KUKA KRL program: vw_bn_usr_s.src, vw_bn_usr_s.dat

--- vw_bn_usr_s.src ---
&ACCESS RV
&REL 11
&COMMENT KS_1.0
&PARAM DISKPATH = KRC:\R1\VW_User\Applikation\Blindnietmuttern
&PARAM TPVW_VERSION = 8.1.8
DEF vw_bn_usr_s( )
;FOLD Aenderungsjournal
;*-------------------------------------------------*
;*Technologiepaket Blindnietmuttern                *
;*                                                 *
;*Konzernstandard                                  *
;*Bearbeiter: B.Mildenberger PEF-2/E0A             *
;*                                                 *
;* Erstellt am:                                    *
;* 2016.02.19 BM                                   *
;*                                                 *
;* Aenderungsjournal                               *
;*                                                 *
;*-------------------------------------------------*
;ENDFOLD Aenderungsjournal
END
;
;FOLD INIT Blindnietmuttern
GLOBAL DEF BN_INIT( )
INT i
;
;FOLD Version Techpaket
Tech_BN.Name[]="KS24.01.002_160220"
;ENDFOLD
;
;FOLD Vorbesetzung Meldungsausgabe
FOR I = 1 TO 100
  n_BN_Handle[I]=-1
ENDFOR
;ENDFOLD
;
$OUT[O_BN_StartPrz[1]]=FALSE
;
END
;ENDFOLD
;
;---------------------------------------------------
;FOLD SAW Blindnietmuttern
GLOBAL DEF BN_SAW( )
INT i
;
;
END
;ENDFOLD
;
;---------------------------------------------------
;FOLD RESET Blindnietmuttern
GLOBAL DEF BN_RESET( )
INT i
;
$OUT[O_BN_StartPrz[1]]=FALSE
;
END
;ENDFOLD
;
;---------------------------------------------------
;FOLD CANCEL Blindnietmuttern
GLOBAL DEF BN_CANCEL( )
INT i
;
$OUT[O_BN_StartPrz[1]]=FALSE
;
END
;ENDFOLD
;
;---------------------------------------------------
;FOLD LOOP Blindnietmuttern
GLOBAL DEF BN_LOOP()
;
FOR BN_ActApp = 1 TO BN_MaxApp
  IF Mit_BN[BN_ActApp] THEN
    ;FOLD Lebensbit
    BN_lBit(BN_ActApp)
    ;ENDFOLD Lebensbit
;
    ;RESET im Fehlerfall ausloesen
    IF NOT BN_QuitHifu[BN_ActApp] AND (NOT $OUT[O_R_SAK] OR NOT $OUT[O_R_RK100]) THEN
      BN_QuitHifu[BN_ActApp]=TRUE
      ;Anstehende Prozesse sicher beenden
      $OUT[O_BN_Reload[BN_ActApp]]=FALSE
      $OUT[O_BN_StartPrz[BN_ActApp]]=FALSE
    ENDIF
    SWITCH BN1_ErrorCode ;Gezieltes Quittieren selektierter Fehler
	  CASE 107, 108
	    BN_FrgQuitHifu[BN_ActApp]=FALSE;keine Freigabe Autoquit
	  DEFAULT
        BN_FrgQuitHifu[BN_ActApp]=TRUE
	ENDSWITCH
    ;Ruecksetzen Ausgaben nach Fehler
    IF $OUT[O_R_RK100] AND $OUT[O_R_SAK] AND BN_QuitHifu[BN_ActApp] AND BN_FrgQuitHifu[BN_ActApp] AND $COULD_START_MOTION THEN
      $OUT[O_BN_Reset[BN_ActApp]]=TRUE
	  IF (($ROB_TIMER - QuitTimer_BN[BN_ActApp]) > 500) THEN
	    $OUT[O_BN_Init[BN_ActApp]]=TRUE
	    $OUT[O_BN_Reset[BN_ActApp]]=FALSE
		IF $OUT[O_BN_Init[BN_ActApp]] AND $IN[I_BN_FkInit[BN_ActApp]] THEN
  	      $OUT[O_BN_Init[BN_ActApp]]=FALSE
		  BN_QuitHifu[BN_ActApp]=FALSE
	    ELSE
        IF (($ROB_TIMER - QuitTimer_BN[BN_ActApp]) > 5000) AND $IN[I_BN_AUTO[BN_ActApp]] THEN
		    BN_Msg(2,#QuitMsg)
			;Retry Init
			$OUT[O_BN_Reset[BN_ActApp]]=TRUE
			QuitTimer_BN[BN_ActApp] = 0
            QuitTimer_BN[BN_ActApp] = $ROB_TIMER
		  ENDIF
		ENDIF
	  ENDIF
	ELSE
      QuitTimer_BN[BN_ActApp] = 0
      QuitTimer_BN[BN_ActApp] = $ROB_TIMER
    ENDIF
;
    ;BA-Hand an BNx setzen
    IF $OUT[O_R_Hand] AND NOT $COULD_START_MOTION THEN
      $OUT[O_BN_R_Hand[BN_ActApp]]=TRUE
      $OUT[O_BN_R_Auto[BN_ActApp]]=FALSE
    ENDIF
;
    ;BA-AUTO an NZ 1 setzen
    IF ($OUT[O_R_Proz_akt] OR $OUT[O_R_bewegt]) OR $OUT[O_R_Auto] THEN
      $OUT[O_BN_R_Hand[BN_ActApp]]=FALSE
      $OUT[O_BN_R_Auto[BN_ActApp]]=TRUE
    ENDIF
;
    ;Anwahl Energiesparmodus
    $OUT[O_BN_eMode[BN_ActApp]] = (($Brake_Sig==0) AND $timer_flag[TimerNr_E_Mo] AND e_Mode_Hilf2)
    ;Freigabe Steuerluft
    $OUT[O_BN_FrgP[BN_ActApp]] = $IN[I_BD01ND] AND $IN[I_MedVorh]
;
    ;Setzweg fuer Visualisierung in CorrMode
	BN_Setzweg_Act[BN_ActApp]=ABS(BN1_SetzWeg)/10 ;[1/10mm]
;
    ;Ausgabe Fehlermeldungen
;
    ;Nieten n.i.O.
    $OUT[O_BN_PrzNio[BN_ActApp]]=$OUT[O_R_Auto] AND $COULD_START_MOTION AND $OUT[O_BN_P_act[BN_ActApp]] AND $FLAG[F_BN_PrzNiO[BN_ActApp]]
    ;Vorwarnung liegt an
    $OUT[O_BN_VwStdm[BN_ActApp]]=$OUT[O_R_Auto] AND $COULD_START_MOTION AND ($IN[I_BN_WarnZugDorn[BN_ActApp]] OR $IN[I_BN_WarnOel[BN_ActApp]])
    ;Verklemmanzeige
    $OUT[O_BN_Verkl[BN_ActApp]]=$OUT[O_R_Auto] AND $COULD_START_MOTION AND NOT $IN[I_BN_AusglIo[BN_ActApp]]
    ;Startbereit fehlt
    $OUT[O_BN_StartBerFehl[BN_ActApp]]=$OUT[O_R_Auto] AND $COULD_START_MOTION AND NOT $IN[I_BN_Ready[BN_ActApp]] AND $FLAG[F_BN_Sammel[BN_ActApp]] AND $timer_flag[TimerNr_Ein]
    ;Betriebsbereit fehlt
    $OUT[O_BN_BereitFehlt[BN_ActApp]]=$OUT[O_R_Auto] AND $COULD_START_MOTION AND NOT $IN[I_BN_Ready[BN_ActApp]] AND $timer_flag[TimerNr_Ein]
    ;Sammelstoerung
    $OUT[O_BN_Sammel[BN_ActApp]]=$OUT[O_R_Auto] AND $COULD_START_MOTION AND ($FLAG[F_BN_Sammel[BN_ActApp]] OR $IN[I_BN_Sammel[BN_ActApp]] OR BN_LBitFeh[BN_ActApp] OR $IN[I_BN_StdmZugDorn[BN_ActApp]]) AND $timer_flag[TimerNr_Ein]
    ;Stoerung quittieren
	IF (BN_ActApp==1) THEN
 	  BN_ErrorCodeAct[1]=BN1_ErrorCode
	ENDIF
	SWITCH BN1_ErrorCode ;Vorhaltung zur gezielten Reaktion auf bestimmte Fehleransprachen
	  CASE 0
	    ;löppt
	  CASE 108 ; Fehler Zugdorn darf nicht via Panel quittiert werden
	    ;#dummy
	  DEFAULT
        $OUT[O_BN_Reset[BN_ActApp]]= $IN[I_BN_Sammel[BN_ActApp]] AND $IN[I_BN_AnwZ1[BN_ActApp]] AND $IN[I_R_Quit_Wei]
	ENDSWITCH
;
    ;Ausgabe Zangencode
    IF NOT Docking THEN
      BN1_ZCode=1
    ENDIF
;
  ENDIF
ENDFOR
;
;ENDFOLD
END
;ENDFOLD
;
;---------------------------------------------------
;---------------------------------------------------
;FOLD Blindnietmuttern_Meldungen
DEF BN_Msg(msg_nr :IN, MsgTyp :IN)
INT msg_nr, Answer
DECL BN_MsgType MsgTyp
DECL KrlMsg_T USER_MSG
DECL KrlMsgPar_T Par[3]
DECL KrlMsgOpt_T Opt
;
USER_MSG = { Modul[] "BN_S_Msg", Nr -1, Msg_txt[] " "}
Opt = { VL_Stop FALSE, Clear_P_Reset TRUE, Log_To_DB TRUE }
Par[1] = { Par_type #Value, Par_txt[] " " }
;
;
IF ((n_BN_Handle[msg_nr]<0) OR (MsgTyp==#NotifyMsg) OR (MsgTyp==#QuitMsg)) THEN
  USER_MSG.Nr = msg_nr
  SWITCH msg_nr
    CASE 1
	   USER_MSG.MSG_TXT[]="Blindnietmutternsteuerung Lebensbitfehler"
    CASE 2
	   USER_MSG.MSG_TXT[]="Initialisierungsfehler Blindnietmutternsteuerung"
    DEFAULT
	   USER_MSG.MSG_TXT[]="unbekannte Meldung"
  ENDSWITCH
  SWITCH MsgTyp
    CASE #StateMsg
      n_BN_Handle[msg_nr] = Set_KrlMsg (#State, USER_MSG, Par[], Opt) ;Ausgabe Statusmeldung
    CASE #QuitMsg
      n_BN_Handle[msg_nr] = Set_KrlMsg (#Quit, USER_MSG, Par[], Opt) ;Ausgabe Quittierungsmeldung
    CASE #NotifyMsg
      n_BN_Handle[msg_nr] = Set_KrlMsg (#Notify, USER_MSG, Par[], Opt) ;Ausgabe Hinweismeldung
    DEFAULT
      n_BN_Handle[msg_nr] = Set_KrlMsg (#Quit, USER_MSG, Par[], Opt) ;Ausgabe Quittierungsmeldung
  ENDSWITCH
ENDIF
END
;
;ENDFOLD (Blindnietmuttern Meldungen)
;
;---------------------------------------------------
;FOLD Lebensbit Blindnietmuttern
DEF BN_lBit(AppNr:IN)
BOOL LBitBZ1, bRet
INT AppNr

BN_LBitFeh[AppNr]=FALSE
;Setzen - Rucksetzen Lebensbit Roboter
$OUT[O_BN_LBitRobBn[AppNr]]=NOT $IN[I_BN_LBitBnRob[AppNr]]
;Pruefen Lebensbit von BZ1
IF $IN[I_BN_LBitBnRob[AppNr]]==FALSE THEN
  IF LBitBnRem[AppNr]==FALSE THEN
    TimerNr_BN[AppNr]=$ROB_TIMER
  ENDIF
  LBitBnRem[AppNr]=TRUE
ELSE
  IF LBitBnRem[AppNr]==TRUE THEN
    TimerNr_BN[AppNr]=$ROB_TIMER
  ENDIF
  LBitBnRem[AppNr]=FALSE
ENDIF
;
IF ($ROB_TIMER - TimerNr_BN[AppNr]) > 5000 THEN
  BN_LBitFeh[AppNr]=TRUE
ENDIF
;
IF BN_LBitFeh[AppNr] THEN
  BN_Msg(1,#StateMsg)
ELSE
  BN_LBitFeh[AppNr]=FALSE
ENDIF
END
;ENDFOLD Lebensbit Blindnietmuttern
;

--- vw_bn_usr_s.dat ---
&ACCESS  RV
&COMMENT KS_1.0
&PARAM DISKPATH = VW_User/Applikation/Blindnietmuttern
&PARAM TPVW_VERSION = 8.1.8
&REL 11
DEFDAT  vw_bn_usr_s PUBLIC
;
;*-------------------------------------------------*
;*Technologiepaket Blindnietmuttern                *
;*                                                 *
;*Konzernstandard                                  *
;*Bearbeiter: B.Mildenberger PEF-2/E0A             *
;*                                                 *
;* Erstellt am:                                    *
;* 2016.02.19 BM                                   *
;*                                                 *
;* Aenderungsjournal                               *
;*                                                 *
;*-------------------------------------------------*
;
;FOLD USER_Version
STRUC _Tech_BN CHAR Name[20],INT Datum
DECL _Tech_BN Tech_BN
;ENDFOLD USER_VERSION
;
;FOLD Vorwahlen
GLOBAL BOOL MIT_BN[1]
MIT_BN[1]=FALSE
;ENDFOLD Vorwahlen
;
;FOLD Stukturen
;
;ENDFOLD Strukturen
;
;FOLD Flags
GLOBAL INT F_m_BN[1]
F_m_BN[1]=422
;ENDFOLD FLAGS
;
;FOLD BOOLEAN
;
GLOBAL BOOL LBitBnRem[1]
LBitBnRem[1]=TRUE
GLOBAL BOOL BN_LBitFeh[1]
BN_LBitFeh[1]=FALSE
GLOBAL BOOL BN_QuitHifu[1]
BN_QuitHifu[1]=FALSE
GLOBAL BOOL BN_FrgQuitHifu[1]
BN_FrgQuitHifu[1]=TRUE
;
;ENDFOLD BOOLEAN
;
;FOLD INTEGER
GLOBAL INT F_BN_Sammel[1]
F_BN_Sammel[1]=423
GLOBAL INT F_BN_PrzNiO[1]
F_BN_PrzNiO[1]=424
;
GLOBAL INT I_BN_Ready[1]
I_BN_Ready[1]=1185
GLOBAL INT I_BN_LBitBnRob[1]
I_BN_LBitBnRob[1]=1187
GLOBAL INT I_BN_eMode[1]
I_BN_eMode[1]=1188
GLOBAL INT I_BN_Hand[1]
I_BN_Hand[1]=1189
GLOBAL INT I_BN_Auto[1]
I_BN_Auto[1]=1190
GLOBAL INT I_BN_FkInit[1]
I_BN_FkInit[1]=1191
GLOBAL INT I_BN_FkPrz[1]
I_BN_FkPrz[1]=1193
GLOBAL INT I_BN_PrzIo[1]
I_BN_PrzIo[1]=1194
GLOBAL INT I_BN_Loaded[1]
I_BN_Loaded[1]=1195
GLOBAL INT I_BN_AusglIo[1]
I_BN_AusglIo[1]=1196
GLOBAL INT I_BN_LagVerr[1]
I_BN_LagVerr[1]=1197
GLOBAL INT I_BN_ElemInFd[1]
I_BN_ElemInFd[1]=1200
GLOBAL INT I_BN_ZCodNio[1]
I_BN_ZCodNio[1]=1201
GLOBAL INT I_BN_GCodW1[1]
I_BN_GCodW1[1]=1206
GLOBAL INT I_BN_GCodW2[1]
I_BN_GCodW2[1]=1207
GLOBAL INT I_BN_GCodW4[1]
I_BN_GCodW4[1]=1208
GLOBAL INT I_BN_WarnTopf[1]
I_BN_WarnTopf[1]=1209
GLOBAL INT I_BN_WarnBunker[1]
I_BN_WarnBunker[1]=1210
GLOBAL INT I_BN_WarnZugDorn[1]
I_BN_WarnZugDorn[1]=1211
GLOBAL INT I_BN_StdmZugDorn[1]
I_BN_StdmZugDorn[1]=1212
GLOBAL INT I_BN_BehVoll[1]
I_BN_BehVoll[1]=1213
GLOBAL INT I_BN_WarnOel[1]
I_BN_WarnOel[1]=1214
GLOBAL INT I_BN_Sammel[1]
I_BN_Sammel[1]=1216
;
GLOBAL INT I_BN_OhnePrz[1]
I_BN_OhnePrz[1]=193
GLOBAL INT I_BN_AnwZ1[1]
I_BN_AnwZ1[1]=196
GLOBAL INT I_BN_AnwZ2[1]
I_BN_AnwZ2[1]=197
GLOBAL INT I_BN_AnwZ3[1]
I_BN_AnwZ3[1]=198
GLOBAL INT I_BN_AnwZ4[1]
I_BN_AnwZ4[1]=199
;
GLOBAL INT O_BN_Reset[1]
O_BN_Reset[1]=1185
GLOBAL INT O_BN_LBitRobBn[1]
O_BN_LBitRobBn[1]=1187
GLOBAL INT O_BN_eMode[1]
O_BN_eMode[1]=1188
GLOBAL INT O_BN_R_Hand[1]
O_BN_R_Hand[1]=1189
GLOBAL INT O_BN_R_Auto[1]
O_BN_R_Auto[1]=1190
GLOBAL INT O_BN_Init[1]
O_BN_Init[1]=1191
GLOBAL INT O_BN_FrgPrz[1]
O_BN_FrgPrz[1]=1192
GLOBAL INT O_BN_StartPrz[1]
O_BN_StartPrz[1]=1193
GLOBAL INT O_BN_Ausspind[1]
O_BN_Ausspind[1]=1194
GLOBAL INT O_BN_Reload[1]
O_BN_Reload[1]=1195
GLOBAL INT O_BN_FrgP[1]
O_BN_FrgP[1]=1196
GLOBAL INT O_BN_LagVerr[1]
O_BN_LagVerr[1]=1197
GLOBAL INT O_BN_AnfReload[1]
O_BN_AnfReload[1]=1198
GLOBAL INT O_BN_MS1V1_BT[1]
O_BN_MS1V1_BT[1]=1199
GLOBAL INT O_BN_MS1V2_FD[1]
O_BN_MS1V2_FD[1]=1200
GLOBAL INT O_BN_ZCodW1[1]
O_BN_ZCodW1[1]=1201
GLOBAL INT O_BN_ZCodW2[1]
O_BN_ZCodW2[1]=1202
GLOBAL INT O_BN_ZCodW4[1]
O_BN_ZCodW4[1]=1203
GLOBAL INT O_BN_ZCodRes[1]
O_BN_ZCodRes[1]=1204
;
GLOBAL INT O_BN_P_act[1]
O_BN_P_act[1]=193
GLOBAL INT O_BN_PrzNio[1]
O_BN_PrzNio[1]=195
GLOBAL INT O_BN_VwStdm[1]
O_BN_VwStdm[1]=196
GLOBAL INT O_BN_Verkl[1]
O_BN_Verkl[1]=197
GLOBAL INT O_BN_StartBerFehl[1]
O_BN_StartBerFehl[1]=198
GLOBAL INT O_BN_BereitFehlt[1]
O_BN_BereitFehlt[1]=199
GLOBAL INT O_BN_Sammel[1]
O_BN_Sammel[1]=200
;
GLOBAL INT I_MedVorh=24
GLOBAL INT TimerNr_BN[1]
TimerNr_BN[1]=74950516
GLOBAL INT QuitTimer_BN[1]
QuitTimer_BN[1]=74950517
GLOBAL CONST INT BN_MaxApp=1 ;Schleifenbegrenzung
GLOBAL INT BN_ActApp=2
GLOBAL INT BN_Setzweg_Act[1] ;Setzweg fuer Visualisierung
BN_Setzweg_Act[1]=0
GLOBAL INT BN_ErrorCodeAct[1] ;Fehlercode fuer Visualisierung
BN_ErrorCodeAct[1]=1
;ENDFOLD INTEGER
;
;FOLD REALS
;
;ENDFOLD REALS
;
;FOLD SIGNALS
;Fehlercode
SIGNAL BN1_ErrorCode $IN[1217]  TO $IN[1232]
;Uebergabe Setzweg von BN1
SIGNAL BN1_SetzWeg $IN[1233]  TO $IN[1248]
;Uebergabe Zangencode an BN1
SIGNAL BN1_ZCode $OUT[1201]  TO $OUT[1203]
;ENDFOLD SIGNALS
;
;FOLD Meldungsausgabe
ENUM BN_MsgType StateMsg,QuitMsg,NotifyMsg
GLOBAL INT n_BN_Handle[100]
INT nMsgNum=0
INT RemMsgNum=0
;ENDFOLD

ENDDAT
